TYPE ST_ProductHandlingSysPar :
STRUCT
	GantryA						: ST_GantrySysPar;
	GantryB						: ST_GantrySysPar;
END_STRUCT
END_TYPE

(* stored: Version 1.1.0.1, ProductVersion 3.1.4020.12
   DUT ST_ProductHandlingSysPar: Id {2e3a68e4-b26f-4048-a945-e6a9ee2a5638} *)
